FUNCTION_BLOCK FB_MUL_INT (* INT Multiplication *)
  (* Standard: 61499-1-D.1; Classification: Math *)
  (* Version 0.0, 2002-05-22, JHC, Rockwell Automation *)
  (* Compiler header: package fb.rt.math; *)
  (* Compiler classdef: class FB_MUL_INT extends FBFunction2 *)
  (* Compiler Java IBM VisualAge 3.0 *)
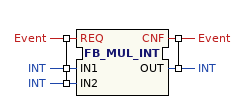
  EVENT_INPUT
    REQ WITH IN1, IN2;
  END_EVENT
  EVENT_OUTPUT
    CNF WITH OUT;
  END_EVENT
  VAR_INPUT
    IN1 : INT; (* Multiplicand *)
    IN2 : INT; (* Multiplier *)
  END_VAR
  VAR_OUTPUT
    OUT : INT; (* Product *)
  END_VAR
END_FUNCTION_BLOCK
